// TIA Portal V21 export
TYPE "Std_Sorgente"
   STRUCT
      Sorgente : Array[0..100] of "Std_Destinazioni";
   END_STRUCT;
END_TYPE
